INTERFACE I_ManualControl

METHOD M_RunPump : BOOL
VAR_INPUT
	bStart : BOOL;
	NTimes : INT;
END_VAR
END_METHOD

METHOD M_RunValve : BOOL
VAR_INPUT
	bStart : BOOL;
END_VAR
END_METHOD

END_INTERFACE

(* stored: Version 1.1.0.1, ProductVersion 3.1.4024.6
   Itf I_ManualControl: Id {45a4907c-dc70-4978-8b7a-d2fa2733690e}
   Method M_RunPump: Id {382576b9-a992-4a6d-adc8-e3eaff8bc674}
   Method M_RunValve: Id {a8996780-dd86-413d-9995-90f1268bfcd4} *)
